FUNCTION_BLOCK PUBLIC ConcreteLoadCell EXTENDS AbstractLoadCell
VAR_INPUT
END_VAR
VAR_OUTPUT
END_VAR
VAR
END_VAR

END_FUNCTION_BLOCK

(* stored: Version 1.1.0.1, ProductVersion 3.1.4024.12
   POU ConcreteLoadCell: Id {7ae39fc0-1d4f-4f20-aec2-7272e61a71f8}, SpecialFunc None *)
